Omron CX-Programmer project NuovoProgetto (CX-Programmer 9.81)

# PLC ZitiPLC: CJ2M CPU32
I/O table (CPU CJ2M-CPU32): rack 0 slot 0 CJ1W-OD212; rack 0 slot 11 CJ2M-EIP21

## Global symbols (name address type ; comment)
0.00 BOOL  ; Luce verde
0.01 BOOL  ; Luce gialla
0.02 BOOL  ; Luce rossa
0.03 BOOL  ; Sirena
T0000 BOOL  ; Timer luce verde
T0001 BOOL  ; Timer luce gialla
T0002 BOOL  ; Timer luce rossa
T0003 BOOL  ; Timer sirena
W0.00 BOOL  ; Richiesta luce verde
W0.01 BOOL  ; Richiesta luce gialla
W0.02 BOOL  ; Richiesta luce rossa
W0.03 BOOL  ; Richiesta sirena

## Program ZitiPLC_Program (cyclic task 0)

### Section Luci

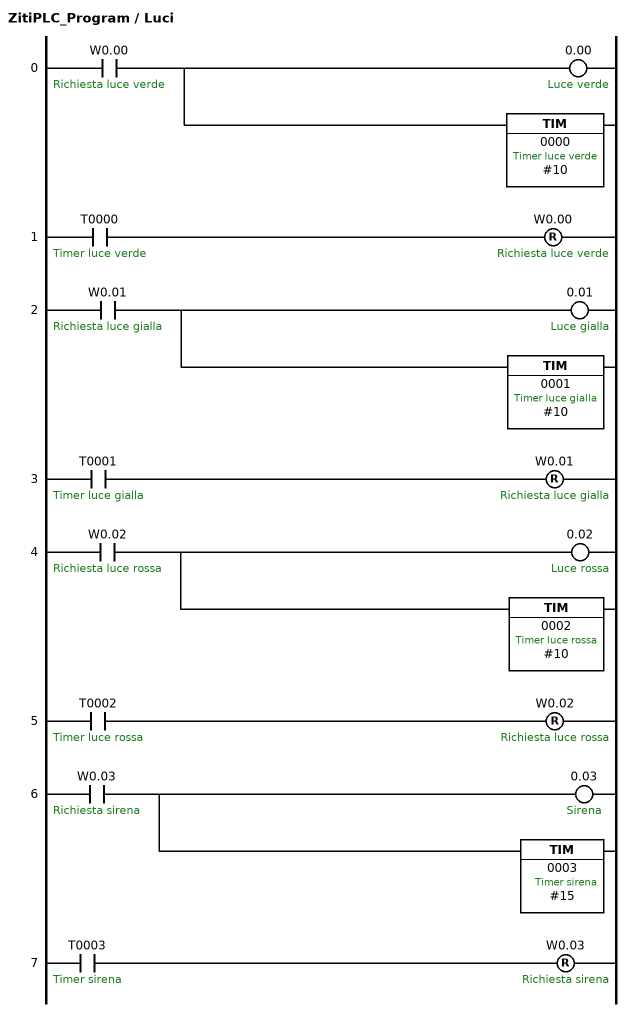
; rung 0
LD W0.00  ; Richiesta luce verde
OUT 0.00  ; Luce verde
TIM 0000 #10  ; Timer luce verde
; rung 1
LD T0000  ; Timer luce verde
RSET W0.00  ; Richiesta luce verde
; rung 2
LD W0.01  ; Richiesta luce gialla
OUT 0.01  ; Luce gialla
TIM 0001 #10  ; Timer luce gialla
; rung 3
LD T0001  ; Timer luce gialla
RSET W0.01  ; Richiesta luce gialla
; rung 4
LD W0.02  ; Richiesta luce rossa
OUT 0.02  ; Luce rossa
TIM 0002 #10  ; Timer luce rossa
; rung 5
LD T0002  ; Timer luce rossa
RSET W0.02  ; Richiesta luce rossa
; rung 6
LD W0.03  ; Richiesta sirena
OUT 0.03  ; Sirena
TIM 0003 #15  ; Timer sirena
; rung 7
LD T0003  ; Timer sirena
RSET W0.03  ; Richiesta sirena

### Section END
; rung 0
END(001)